// SIMATIC S7-200 project (STEP 7-Micro/WIN), CPU 221 REL 01.10

SYMBOL_TABLE USER1
start_btn        I0.0     // start
stop_btn         I0.1     // stop
x1               Q0.0     // xanh 1
v1               Q0.1     // vang 1
d1               Q0.2     // do 1
x2               Q0.3     // xanh 2
v2               Q0.4     // vang 2
d2               Q0.5     // do 2
en_time1         M0.1     // enable timer 1
en_time2         M0.2     // enable timer 2
en_time3         M0.3     // enable timer 3
en_time4         M0.4     // enable timer 4
END_SYMBOL_TABLE

ORGANIZATION_BLOCK MAIN:OB1
TITLE=PROGRAM COMMENTS
BEGIN
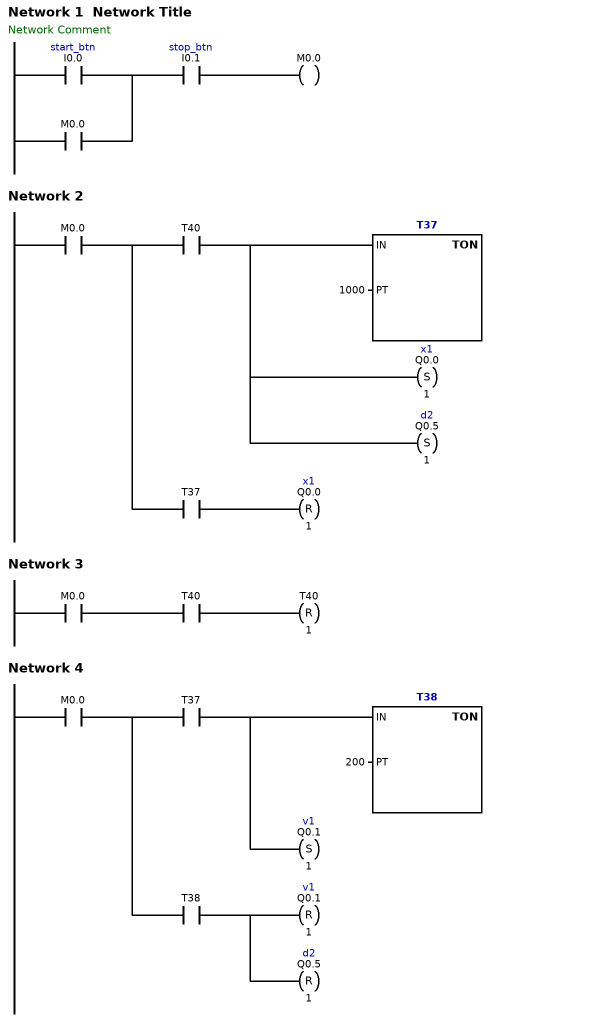
Network 1 // Network Title
// Network Comment
LD     start_btn:I0.0
O      M0.0
A      stop_btn:I0.1
=      M0.0
Network 2
// (network saved uncompiled; LAD cells follow)
// row 0: c0 -| |- M0.0 v  c1 -| |- T40 v  c2 --  c3 [TON T37 IN:=power@row0, PT:=1000]
// row 1: c0 ^v  c1 ^v  c3 [box]
// row 2: c0 ^v  c1 ^v  c2 --  c3 -(S) x1:Q0.0, 1
// row 3: c0 ^v  c1 ^  c2 --  c3 -(S) d2:Q0.5, 1
// row 4: c0 ^  c1 -| |- T37  c2 -(R) x1:Q0.0, 1
Network 3
// (network saved uncompiled; LAD cells follow)
// row 0: c0 -| |- M0.0  c1 -| |- T40  c2 -(R) T40, 1
Network 4
// (network saved uncompiled; LAD cells follow)
// row 0: c0 -| |- M0.0 v  c1 -| |- T37 v  c2 --  c3 [TON T38 IN:=power@row0, PT:=200]
// row 1: c0 ^v  c1 ^v  c3 [box]
// row 2: c0 ^v  c1 ^  c2 -(S) v1:Q0.1, 1
// row 3: c0 ^  c1 -| |- T38 v  c2 -(R) v1:Q0.1, 1
// row 4: c1 ^  c2 -(R) d2:Q0.5, 1
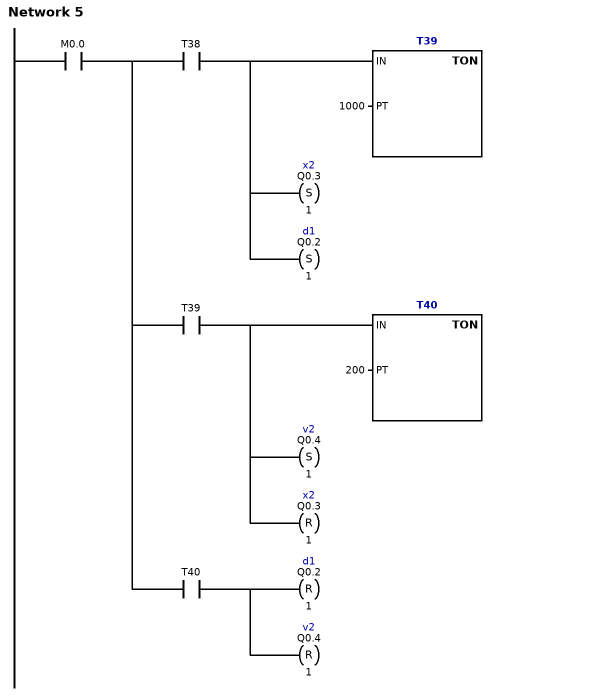
Network 5
// (network saved uncompiled; LAD cells follow)
// row 0: c0 -| |- M0.0 v  c1 -| |- T38 v  c2 --  c3 [TON T39 IN:=power@row0, PT:=1000]
// row 1: c0 ^v  c1 ^v  c3 [box]
// row 2: c0 ^v  c1 ^v  c2 -(S) x2:Q0.3, 1
// row 3: c0 ^v  c1 ^  c2 -(S) d1:Q0.2, 1
// row 4: c0 ^v  c1 -| |- T39 v  c2 --  c3 [TON T40 IN:=power@row4, PT:=200]
// row 5: c0 ^v  c1 ^v  c3 [box]
// row 6: c0 ^v  c1 ^v  c2 -(S) v2:Q0.4, 1
// row 7: c0 ^v  c1 ^  c2 -(R) x2:Q0.3, 1
// row 8: c0 ^  c1 -| |- T40 v  c2 -(R) d1:Q0.2, 1
// row 9: c1 ^  c2 -(R) v2:Q0.4, 1
END_ORGANIZATION_BLOCK
